// LS Electric XG5000 project: SPAV_PANEL
// PLC LSPLC

PROGRAM 00MAIN (task: 스캔 프로그램)

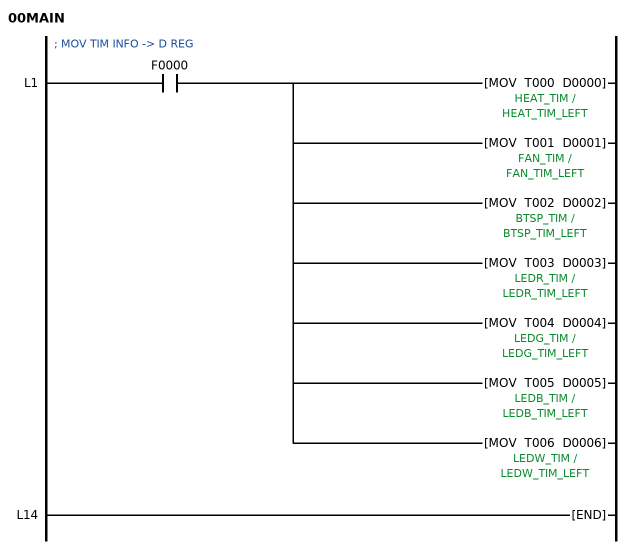
// MOV TIM INFO -> D REG
; L1
LOAD      F0000
MOV       T000 D0000	// HEAT_TIM / HEAT_TIM_LEFT
MOV       T001 D0001	// FAN_TIM / FAN_TIM_LEFT
MOV       T002 D0002	// BTSP_TIM / BTSP_TIM_LEFT
MOV       T003 D0003	// LEDR_TIM / LEDR_TIM_LEFT
MOV       T004 D0004	// LEDG_TIM / LEDG_TIM_LEFT
MOV       T005 D0005	// LEDB_TIM / LEDB_TIM_LEFT
MOV       T006 D0006	// LEDW_TIM / LEDW_TIM_LEFT
; L14
END

PROGRAM 01INPUT (task: 스캔 프로그램)

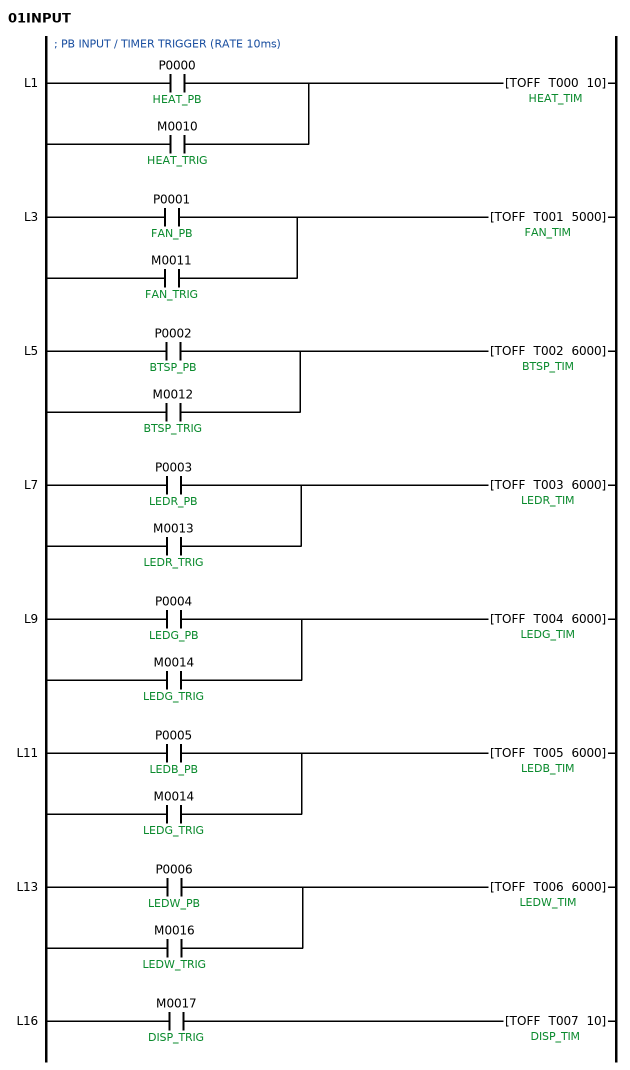
// PB INPUT / TIMER TRIGGER (RATE 10ms)
; L1
LOAD      P0000	// HEAT_PB
OR        M0010	// HEAT_TRIG
TOFF      T000 10	// HEAT_TIM
; L3
LOAD      P0001	// FAN_PB
OR        M0011	// FAN_TRIG
TOFF      T001 5000	// FAN_TIM
; L5
LOAD      P0002	// BTSP_PB
OR        M0012	// BTSP_TRIG
TOFF      T002 6000	// BTSP_TIM
; L7
LOAD      P0003	// LEDR_PB
OR        M0013	// LEDR_TRIG
TOFF      T003 6000	// LEDR_TIM
; L9
LOAD      P0004	// LEDG_PB
OR        M0014	// LEDG_TRIG
TOFF      T004 6000	// LEDG_TIM
; L11
LOAD      P0005	// LEDB_PB
OR        M0014	// LEDG_TRIG
TOFF      T005 6000	// LEDB_TIM
; L13
LOAD      P0006	// LEDW_PB
OR        M0016	// LEDW_TRIG
TOFF      T006 6000	// LEDW_TIM
; L16
LOAD      M0017	// DISP_TRIG
TOFF      T007 10	// DISP_TIM

PROGRAM 02OUTPUT (task: 스캔 프로그램)

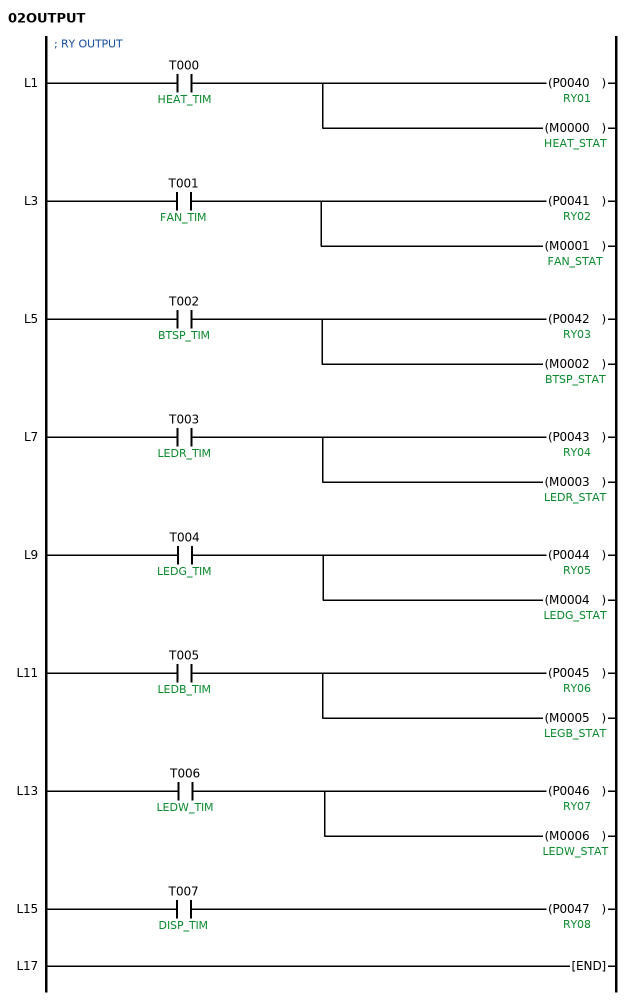
// RY OUTPUT
; L1
LOAD      T000	// HEAT_TIM
OUT       P0040	// RY01
OUT       M0000	// HEAT_STAT
; L3
LOAD      T001	// FAN_TIM
OUT       P0041	// RY02
OUT       M0001	// FAN_STAT
; L5
LOAD      T002	// BTSP_TIM
OUT       P0042	// RY03
OUT       M0002	// BTSP_STAT
; L7
LOAD      T003	// LEDR_TIM
OUT       P0043	// RY04
OUT       M0003	// LEDR_STAT
; L9
LOAD      T004	// LEDG_TIM
OUT       P0044	// RY05
OUT       M0004	// LEDG_STAT
; L11
LOAD      T005	// LEDB_TIM
OUT       P0045	// RY06
OUT       M0005	// LEGB_STAT
; L13
LOAD      T006	// LEDW_TIM
OUT       P0046	// RY07
OUT       M0006	// LEDW_STAT
; L15
LOAD      T007	// DISP_TIM
OUT       P0047	// RY08
; L17
END

VARIABLES AND COMMENTS (devices not used above)
M00015	BIT	LEDB_TRIG
P00048	BIT	RY09